// TwinCAT 3 PLC project Example
// ProgramVersion: 3.1.4026.19
// libraries:
//   TAC_Events, * (Timberline Automation and Control Co.)
//   Tc2_Standard, * (Beckhoff Automation GmbH)
//   Tc2_System, * (Beckhoff Automation GmbH)
// project tree:
//   / PlcTask.TcTTO
//   POUs/ Example.TcPOU
// (motion and I/O tree: see PLC project tac_events)
// real-time tasks:
//   TASK PlcTask: cycle T#10ms, priority 20, ADS port 350
//   TASK PlcTask1: cycle T#10ms, priority 21, ADS port 351

CONFIGURATION Example
    RESOURCE PLC ON TwinCAT3
        TASK PlcTask(INTERVAL := T#10ms, PRIORITY := 21);
        PROGRAM Example WITH PlcTask : Example;
    END_RESOURCE
END_CONFIGURATION

// ---- POUs/Example.TcPOU
PROGRAM Example
VAR
	init : BOOL := TRUE;
	logMsg : STRING;
	logger : T_Logger;
	
	
	triggerInfo : BOOL;
	triggerWarning : BOOL;
	triggerError : BOOL;
	triggerCritical : BOOL;
	
	
	
END_VAR

IF init THEN
	TAC_Events.LogConfig.LogLevel := E_LogSeverity.Debug;
	init := FALSE;
END_IF

IF triggerInfo THEN
    logMsg := 'Test Info of Logger';
    logger.LogInfo(logMsg);
    triggerInfo := FALSE;
END_IF

IF triggerWarning THEN
    logMsg := 'Test Warning of Logger';
    logger.LogWarning(logMsg);
    triggerWarning := FALSE;
END_IF

IF triggerError THEN
    logMsg := 'Test Error of Logger';
    logger.LogError(logMsg);
    triggerError := FALSE;
END_IF

IF triggerCritical THEN
    logMsg := 'Test Critical of Logger';
    logger.LogCritical(logMsg);
    triggerCritical := FALSE;
END_IF

END_PROGRAM
